// TIA Portal V17 export
// export: Created 2024-08-07T21:44:17.5349337Z, ExportSetting WithDefaults, DisplayName Totally Integrated Automation Portal, DisplayVersion V17 Update 7, DisplayName TIA Portal Openness, DisplayVersion V17 Update 7, DisplayName TIA Portal Version Control Interface, DisplayVersion V17, DisplayName SINAMICS Startdrive Advanced, DisplayVersion V17 SP2, DisplayName SINAMICS Startdrive G110M, G120, G120C, G120D, G120P, G115D, DisplayVersion V17 SP2, DisplayName SINAMICS Startdrive G130, G150, S120, S150, SINAMICS MV, S210, DisplayVersion V17 SP2, DisplayName STEP 7 Professional, DisplayVersion V17 Update 7, DisplayName STEP 7 Safety, DisplayVersion V17 Update 6, DisplayName WinCC Advanced / Unified PC, DisplayVersion V17 Update 7
TYPE "typeOpcUaAllowedDataTypes"
// stored: IsFailsafeCompliant false
   STRUCT
      "bool" : Bool;   // Maps to Boolean
      sInt : SInt;   // Maps to SByte
      "int" : Int;   // Maps to Int16
      "dInt" : DInt;   // Maps to Int32
      lInt : LInt;   // Maps to Int64
      uSInt : USInt;   // Maps to Byte
      uInt : UInt;   // Maps to Uint16
      uDInt : UDInt;   // Maps to Uint32
      uLInt : ULInt;   // Maps to Uint64
      "real" : Real;   // Maps to Float
      lReal : LReal;   // Maps to Double
      ldt : LDT;   // Maps to DateTime
      wString : WString;   // Maps to String
      opcUaNodeId { S7_SetPoint := 'True'} : OPC_UA_NodeId;
      opcUaQualifiedName { S7_SetPoint := 'True'} : OPC_UA_QualifiedName;
      myUnion { S7_SetPoint := 'True'} : "typeUnionMyDatatype";
      locText { S7_SetPoint := 'True'} : "typeOpcUaLocalizedText";
      myByteString { S7_SetPoint := 'True'} : "typeOpcUaByteString";
      guid { S7_SetPoint := 'True'} : "typeOpcUaGuid";
   END_STRUCT;
END_TYPE
